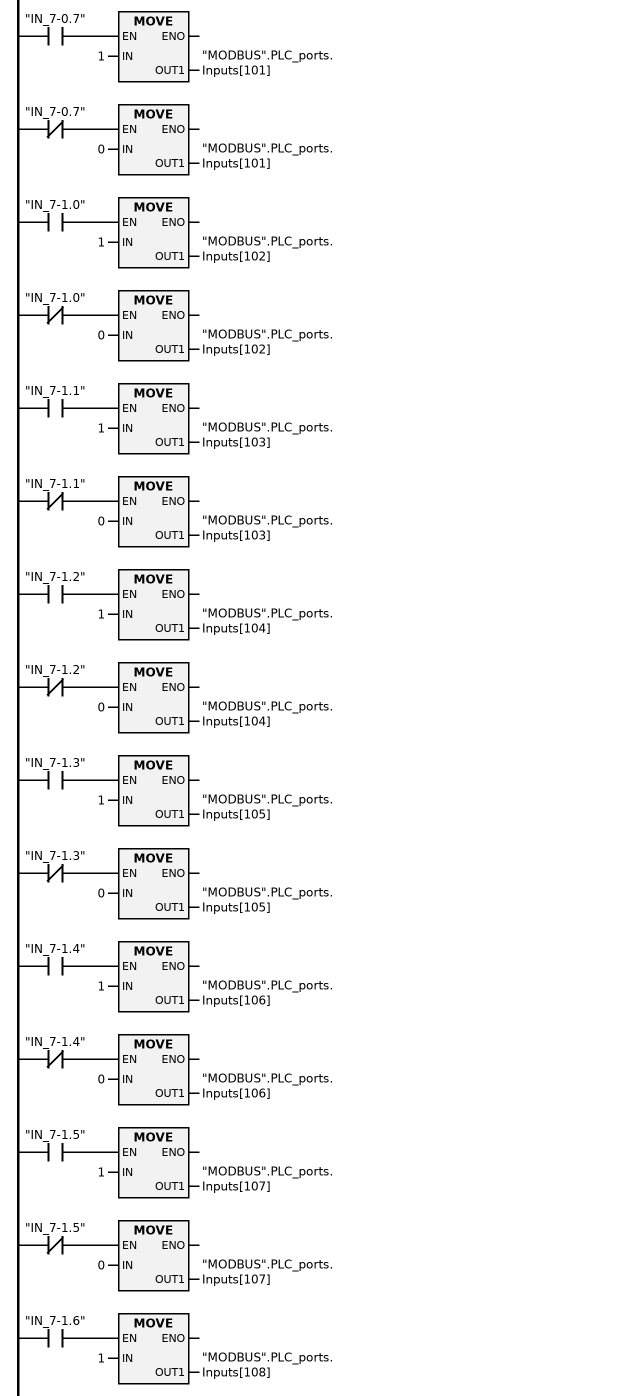
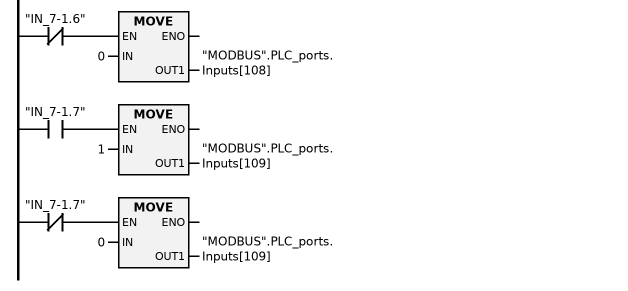
   RUNG wire#powerrail
      Contact( "IN_7-0.0" )
      Move(in := 1, out1 => "MODBUS".PLC_ports.Inputs[94])
   END_RUNG
   RUNG wire#powerrail
      I_Contact( "IN_7-0.0" )
      Move(in := 0, out1 => "MODBUS".PLC_ports.Inputs[94])
   END_RUNG
   RUNG wire#powerrail
      Contact( "IN_7-0.1" )
      Move(in := 1, out1 => "MODBUS".PLC_ports.Inputs[95])
   END_RUNG
   RUNG wire#powerrail
      I_Contact( "IN_7-0.1" )
      Move(in := 0, out1 => "MODBUS".PLC_ports.Inputs[95])
   END_RUNG
   RUNG wire#powerrail
      Contact( "IN_7-0.2" )
      Move(in := 1, out1 => "MODBUS".PLC_ports.Inputs[96])
   END_RUNG
   RUNG wire#powerrail
      I_Contact( "IN_7-0.2" )
      Move(in := 0, out1 => "MODBUS".PLC_ports.Inputs[96])
   END_RUNG
   RUNG wire#powerrail
      Contact( "IN_7-0.3" )
      Move(in := 1, out1 => "MODBUS".PLC_ports.Inputs[97])
   END_RUNG
   RUNG wire#powerrail
      I_Contact( "IN_7-0.3" )
      Move(in := 0, out1 => "MODBUS".PLC_ports.Inputs[97])
   END_RUNG
   RUNG wire#powerrail
      Contact( "IN_7-0.4" )
      Move(in := 1, out1 => "MODBUS".PLC_ports.Inputs[98])
   END_RUNG
   RUNG wire#powerrail
      I_Contact( "IN_7-0.4" )
      Move(in := 0, out1 => "MODBUS".PLC_ports.Inputs[98])
   END_RUNG
   RUNG wire#powerrail
      Contact( "IN_7-0.5" )
      Move(in := 1, out1 => "MODBUS".PLC_ports.Inputs[99])
   END_RUNG
   RUNG wire#powerrail
      I_Contact( "IN_7-0.5" )
      Move(in := 0, out1 => "MODBUS".PLC_ports.Inputs[99])
   END_RUNG
   RUNG wire#powerrail
      Contact( "IN_7-0.6" )
      Move(in := 1, out1 => "MODBUS".PLC_ports.Inputs[100])
   END_RUNG
   RUNG wire#powerrail
      I_Contact( "IN_7-0.6" )
      Move(in := 0, out1 => "MODBUS".PLC_ports.Inputs[100])
   END_RUNG
   RUNG wire#powerrail
      Contact( "IN_7-0.7" )
      Move(in := 1, out1 => "MODBUS".PLC_ports.Inputs[101])
   END_RUNG
   RUNG wire#powerrail
      I_Contact( "IN_7-0.7" )
      Move(in := 0, out1 => "MODBUS".PLC_ports.Inputs[101])
   END_RUNG
   RUNG wire#powerrail
      Contact( "IN_7-1.0" )
      Move(in := 1, out1 => "MODBUS".PLC_ports.Inputs[102])
   END_RUNG
   RUNG wire#powerrail
      I_Contact( "IN_7-1.0" )
      Move(in := 0, out1 => "MODBUS".PLC_ports.Inputs[102])
   END_RUNG
   RUNG wire#powerrail
      Contact( "IN_7-1.1" )
      Move(in := 1, out1 => "MODBUS".PLC_ports.Inputs[103])
   END_RUNG
   RUNG wire#powerrail
      I_Contact( "IN_7-1.1" )
      Move(in := 0, out1 => "MODBUS".PLC_ports.Inputs[103])
   END_RUNG
   RUNG wire#powerrail
      Contact( "IN_7-1.2" )
      Move(in := 1, out1 => "MODBUS".PLC_ports.Inputs[104])
   END_RUNG
   RUNG wire#powerrail
      I_Contact( "IN_7-1.2" )
      Move(in := 0, out1 => "MODBUS".PLC_ports.Inputs[104])
   END_RUNG
   RUNG wire#powerrail
      Contact( "IN_7-1.3" )
      Move(in := 1, out1 => "MODBUS".PLC_ports.Inputs[105])
   END_RUNG
   RUNG wire#powerrail
      I_Contact( "IN_7-1.3" )
      Move(in := 0, out1 => "MODBUS".PLC_ports.Inputs[105])
   END_RUNG
   RUNG wire#powerrail
      Contact( "IN_7-1.4" )
      Move(in := 1, out1 => "MODBUS".PLC_ports.Inputs[106])
   END_RUNG
   RUNG wire#powerrail
      I_Contact( "IN_7-1.4" )
      Move(in := 0, out1 => "MODBUS".PLC_ports.Inputs[106])
   END_RUNG
   RUNG wire#powerrail
      Contact( "IN_7-1.5" )
      Move(in := 1, out1 => "MODBUS".PLC_ports.Inputs[107])
   END_RUNG
   RUNG wire#powerrail
      I_Contact( "IN_7-1.5" )
      Move(in := 0, out1 => "MODBUS".PLC_ports.Inputs[107])
   END_RUNG
   RUNG wire#powerrail
      Contact( "IN_7-1.6" )
      Move(in := 1, out1 => "MODBUS".PLC_ports.Inputs[108])
   END_RUNG
   RUNG wire#powerrail
      I_Contact( "IN_7-1.6" )
      Move(in := 0, out1 => "MODBUS".PLC_ports.Inputs[108])
   END_RUNG
   RUNG wire#powerrail
      Contact( "IN_7-1.7" )
      Move(in := 1, out1 => "MODBUS".PLC_ports.Inputs[109])
   END_RUNG
   RUNG wire#powerrail
      I_Contact( "IN_7-1.7" )
      Move(in := 0, out1 => "MODBUS".PLC_ports.Inputs[109])
   END_RUNG
   // the same network as SCL:
   IF "IN_7-0.0" THEN "MODBUS".PLC_ports.Inputs[94] := 1; END_IF;
   IF NOT "IN_7-0.0" THEN "MODBUS".PLC_ports.Inputs[94] := 0; END_IF;
   IF "IN_7-0.1" THEN "MODBUS".PLC_ports.Inputs[95] := 1; END_IF;
   IF NOT "IN_7-0.1" THEN "MODBUS".PLC_ports.Inputs[95] := 0; END_IF;
   IF "IN_7-0.2" THEN "MODBUS".PLC_ports.Inputs[96] := 1; END_IF;
   IF NOT "IN_7-0.2" THEN "MODBUS".PLC_ports.Inputs[96] := 0; END_IF;
   IF "IN_7-0.3" THEN "MODBUS".PLC_ports.Inputs[97] := 1; END_IF;
   IF NOT "IN_7-0.3" THEN "MODBUS".PLC_ports.Inputs[97] := 0; END_IF;
   IF "IN_7-0.4" THEN "MODBUS".PLC_ports.Inputs[98] := 1; END_IF;
   IF NOT "IN_7-0.4" THEN "MODBUS".PLC_ports.Inputs[98] := 0; END_IF;
   IF "IN_7-0.5" THEN "MODBUS".PLC_ports.Inputs[99] := 1; END_IF;
   IF NOT "IN_7-0.5" THEN "MODBUS".PLC_ports.Inputs[99] := 0; END_IF;
   IF "IN_7-0.6" THEN "MODBUS".PLC_ports.Inputs[100] := 1; END_IF;
   IF NOT "IN_7-0.6" THEN "MODBUS".PLC_ports.Inputs[100] := 0; END_IF;
   IF "IN_7-0.7" THEN "MODBUS".PLC_ports.Inputs[101] := 1; END_IF;
   IF NOT "IN_7-0.7" THEN "MODBUS".PLC_ports.Inputs[101] := 0; END_IF;
   IF "IN_7-1.0" THEN "MODBUS".PLC_ports.Inputs[102] := 1; END_IF;
   IF NOT "IN_7-1.0" THEN "MODBUS".PLC_ports.Inputs[102] := 0; END_IF;
   IF "IN_7-1.1" THEN "MODBUS".PLC_ports.Inputs[103] := 1; END_IF;
   IF NOT "IN_7-1.1" THEN "MODBUS".PLC_ports.Inputs[103] := 0; END_IF;
   IF "IN_7-1.2" THEN "MODBUS".PLC_ports.Inputs[104] := 1; END_IF;
   IF NOT "IN_7-1.2" THEN "MODBUS".PLC_ports.Inputs[104] := 0; END_IF;
   IF "IN_7-1.3" THEN "MODBUS".PLC_ports.Inputs[105] := 1; END_IF;
   IF NOT "IN_7-1.3" THEN "MODBUS".PLC_ports.Inputs[105] := 0; END_IF;
   IF "IN_7-1.4" THEN "MODBUS".PLC_ports.Inputs[106] := 1; END_IF;
   IF NOT "IN_7-1.4" THEN "MODBUS".PLC_ports.Inputs[106] := 0; END_IF;
   IF "IN_7-1.5" THEN "MODBUS".PLC_ports.Inputs[107] := 1; END_IF;
   IF NOT "IN_7-1.5" THEN "MODBUS".PLC_ports.Inputs[107] := 0; END_IF;
   IF "IN_7-1.6" THEN "MODBUS".PLC_ports.Inputs[108] := 1; END_IF;
   IF NOT "IN_7-1.6" THEN "MODBUS".PLC_ports.Inputs[108] := 0; END_IF;
   IF "IN_7-1.7" THEN "MODBUS".PLC_ports.Inputs[109] := 1; END_IF;
   IF NOT "IN_7-1.7" THEN "MODBUS".PLC_ports.Inputs[109] := 0; END_IF;
END_REGION
END_FUNCTION_BLOCK

FUNCTION_BLOCK "Output signals"   // FB3, LAD
{ S7_Optimized_Access := 'TRUE' }
VERSION : 0.1
BEGIN

REGION Network 1
   // Выходы 1 блока, Siemens S7-1200
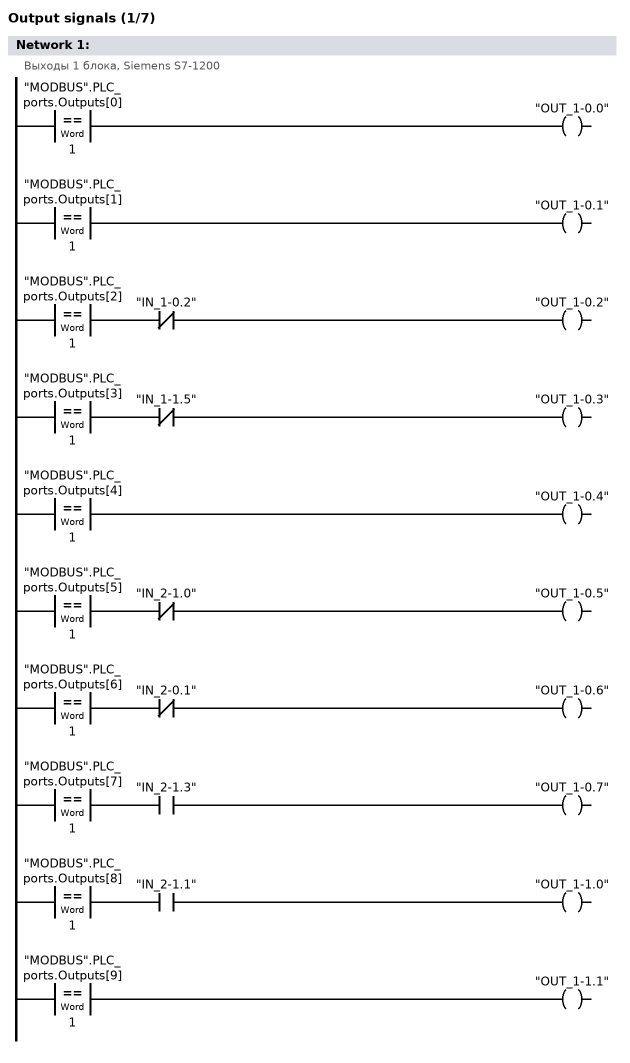
   RUNG wire#powerrail
      { S7_Templates := "SrcType := Word" } EQ_Contact(in1 := "MODBUS".PLC_ports.Outputs[0], in2 := 1)
      Coil( "OUT_1-0.0" )
   END_RUNG
   RUNG wire#powerrail
      { S7_Templates := "SrcType := Word" } EQ_Contact(in1 := "MODBUS".PLC_ports.Outputs[1], in2 := 1)
      Coil( "OUT_1-0.1" )
   END_RUNG
   RUNG wire#powerrail
      { S7_Templates := "SrcType := Word" } EQ_Contact(in1 := "MODBUS".PLC_ports.Outputs[2], in2 := 1)
      I_Contact( "IN_1-0.2" )
      Coil( "OUT_1-0.2" )
   END_RUNG
   RUNG wire#powerrail
      { S7_Templates := "SrcType := Word" } EQ_Contact(in1 := "MODBUS".PLC_ports.Outputs[3], in2 := 1)
      I_Contact( "IN_1-1.5" )
      Coil( "OUT_1-0.3" )
   END_RUNG
   RUNG wire#powerrail
      { S7_Templates := "SrcType := Word" } EQ_Contact(in1 := "MODBUS".PLC_ports.Outputs[4], in2 := 1)
      Coil( "OUT_1-0.4" )
   END_RUNG
   RUNG wire#powerrail
      { S7_Templates := "SrcType := Word" } EQ_Contact(in1 := "MODBUS".PLC_ports.Outputs[5], in2 := 1)
      I_Contact( "IN_2-1.0" )
      Coil( "OUT_1-0.5" )
   END_RUNG
   RUNG wire#powerrail
      { S7_Templates := "SrcType := Word" } EQ_Contact(in1 := "MODBUS".PLC_ports.Outputs[6], in2 := 1)
      I_Contact( "IN_2-0.1" )
      Coil( "OUT_1-0.6" )
   END_RUNG
   RUNG wire#powerrail
      { S7_Templates := "SrcType := Word" } EQ_Contact(in1 := "MODBUS".PLC_ports.Outputs[7], in2 := 1)
      Contact( "IN_2-1.3" )
      Coil( "OUT_1-0.7" )
   END_RUNG
   RUNG wire#powerrail
      { S7_Templates := "SrcType := Word" } EQ_Contact(in1 := "MODBUS".PLC_ports.Outputs[8], in2 := 1)
      Contact( "IN_2-1.1" )
      Coil( "OUT_1-1.0" )
   END_RUNG
   RUNG wire#powerrail
      { S7_Templates := "SrcType := Word" } EQ_Contact(in1 := "MODBUS".PLC_ports.Outputs[9], in2 := 1)
      Coil( "OUT_1-1.1" )
   END_RUNG
   // the same network as SCL:
   "OUT_1-0.0" := "MODBUS".PLC_ports.Outputs[0] = 1;
   "OUT_1-0.1" := "MODBUS".PLC_ports.Outputs[1] = 1;
   "OUT_1-0.2" := ("MODBUS".PLC_ports.Outputs[2] = 1) AND NOT "IN_1-0.2";
   "OUT_1-0.3" := ("MODBUS".PLC_ports.Outputs[3] = 1) AND NOT "IN_1-1.5";
   "OUT_1-0.4" := "MODBUS".PLC_ports.Outputs[4] = 1;
   "OUT_1-0.5" := ("MODBUS".PLC_ports.Outputs[5] = 1) AND NOT "IN_2-1.0";
   "OUT_1-0.6" := ("MODBUS".PLC_ports.Outputs[6] = 1) AND NOT "IN_2-0.1";
   "OUT_1-0.7" := ("MODBUS".PLC_ports.Outputs[7] = 1) AND "IN_2-1.3";
   "OUT_1-1.0" := ("MODBUS".PLC_ports.Outputs[8] = 1) AND "IN_2-1.1";
   "OUT_1-1.1" := "MODBUS".PLC_ports.Outputs[9] = 1;
END_REGION

REGION Network 2
   // Выходы 2 блока, Siemens SM-1223
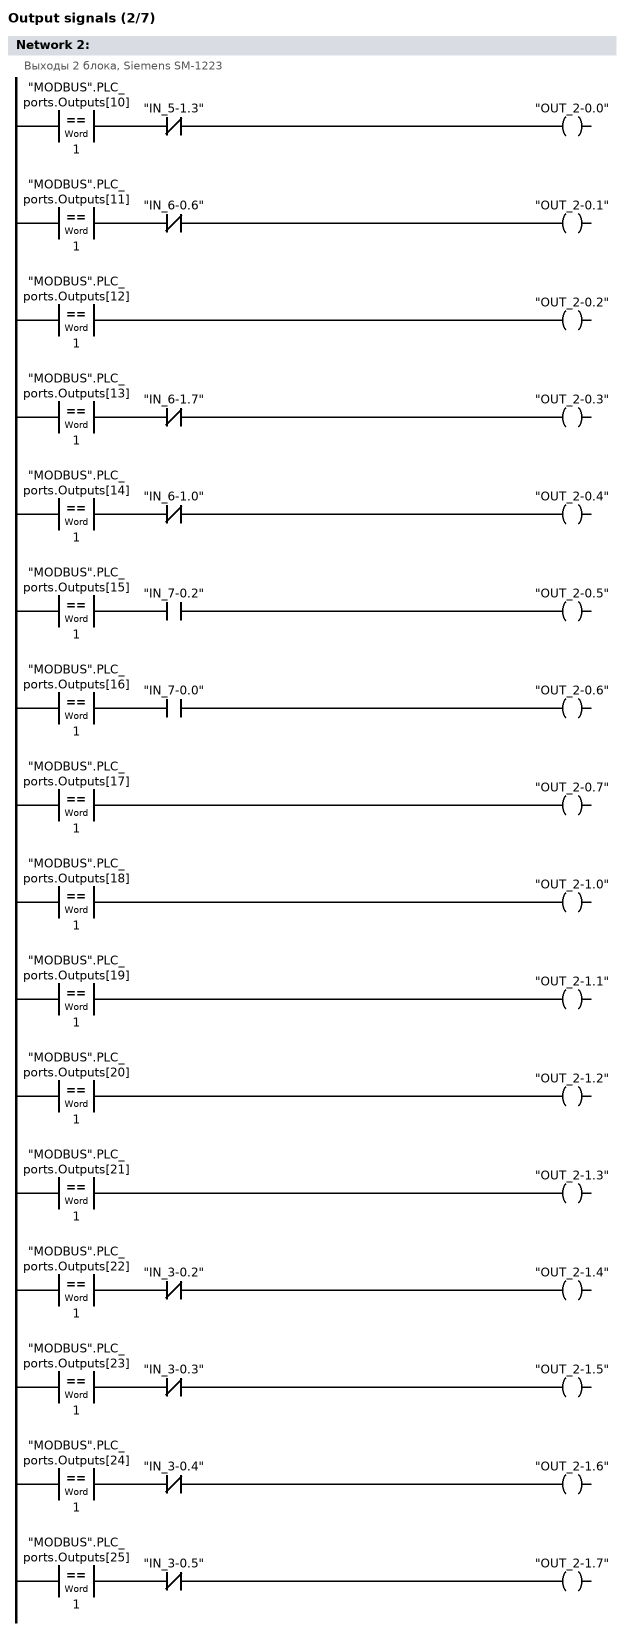
   RUNG wire#powerrail
      { S7_Templates := "SrcType := Word" } EQ_Contact(in1 := "MODBUS".PLC_ports.Outputs[10], in2 := 1)
      I_Contact( "IN_5-1.3" )
      Coil( "OUT_2-0.0" )
   END_RUNG
   RUNG wire#powerrail
      { S7_Templates := "SrcType := Word" } EQ_Contact(in1 := "MODBUS".PLC_ports.Outputs[11], in2 := 1)
      I_Contact( "IN_6-0.6" )
      Coil( "OUT_2-0.1" )
   END_RUNG
   RUNG wire#powerrail
      { S7_Templates := "SrcType := Word" } EQ_Contact(in1 := "MODBUS".PLC_ports.Outputs[12], in2 := 1)
      Coil( "OUT_2-0.2" )
   END_RUNG
   RUNG wire#powerrail
      { S7_Templates := "SrcType := Word" } EQ_Contact(in1 := "MODBUS".PLC_ports.Outputs[13], in2 := 1)
      I_Contact( "IN_6-1.7" )
      Coil( "OUT_2-0.3" )
   END_RUNG
   RUNG wire#powerrail
      { S7_Templates := "SrcType := Word" } EQ_Contact(in1 := "MODBUS".PLC_ports.Outputs[14], in2 := 1)
      I_Contact( "IN_6-1.0" )
      Coil( "OUT_2-0.4" )
   END_RUNG
   RUNG wire#powerrail
      { S7_Templates := "SrcType := Word" } EQ_Contact(in1 := "MODBUS".PLC_ports.Outputs[15], in2 := 1)
      Contact( "IN_7-0.2" )
      Coil( "OUT_2-0.5" )
   END_RUNG
   RUNG wire#powerrail
      { S7_Templates := "SrcType := Word" } EQ_Contact(in1 := "MODBUS".PLC_ports.Outputs[16], in2 := 1)
      Contact( "IN_7-0.0" )
      Coil( "OUT_2-0.6" )
   END_RUNG
   RUNG wire#powerrail
      { S7_Templates := "SrcType := Word" } EQ_Contact(in1 := "MODBUS".PLC_ports.Outputs[17], in2 := 1)
      Coil( "OUT_2-0.7" )
   END_RUNG
   RUNG wire#powerrail
      { S7_Templates := "SrcType := Word" } EQ_Contact(in1 := "MODBUS".PLC_ports.Outputs[18], in2 := 1)
      Coil( "OUT_2-1.0" )
   END_RUNG
   RUNG wire#powerrail
      { S7_Templates := "SrcType := Word" } EQ_Contact(in1 := "MODBUS".PLC_ports.Outputs[19], in2 := 1)
      Coil( "OUT_2-1.1" )
   END_RUNG
   RUNG wire#powerrail
      { S7_Templates := "SrcType := Word" } EQ_Contact(in1 := "MODBUS".PLC_ports.Outputs[20], in2 := 1)
      Coil( "OUT_2-1.2" )
   END_RUNG
   RUNG wire#powerrail
      { S7_Templates := "SrcType := Word" } EQ_Contact(in1 := "MODBUS".PLC_ports.Outputs[21], in2 := 1)
      Coil( "OUT_2-1.3" )
   END_RUNG
   RUNG wire#powerrail
      { S7_Templates := "SrcType := Word" } EQ_Contact(in1 := "MODBUS".PLC_ports.Outputs[22], in2 := 1)
      I_Contact( "IN_3-0.2" )
      Coil( "OUT_2-1.4" )
   END_RUNG
   RUNG wire#powerrail
      { S7_Templates := "SrcType := Word" } EQ_Contact(in1 := "MODBUS".PLC_ports.Outputs[23], in2 := 1)
      I_Contact( "IN_3-0.3" )
      Coil( "OUT_2-1.5" )
   END_RUNG
   RUNG wire#powerrail
      { S7_Templates := "SrcType := Word" } EQ_Contact(in1 := "MODBUS".PLC_ports.Outputs[24], in2 := 1)
      I_Contact( "IN_3-0.4" )
      Coil( "OUT_2-1.6" )
   END_RUNG
   RUNG wire#powerrail
      { S7_Templates := "SrcType := Word" } EQ_Contact(in1 := "MODBUS".PLC_ports.Outputs[25], in2 := 1)
      I_Contact( "IN_3-0.5" )
      Coil( "OUT_2-1.7" )
   END_RUNG
   // the same network as SCL:
   "OUT_2-0.0" := ("MODBUS".PLC_ports.Outputs[10] = 1) AND NOT "IN_5-1.3";
   "OUT_2-0.1" := ("MODBUS".PLC_ports.Outputs[11] = 1) AND NOT "IN_6-0.6";
   "OUT_2-0.2" := "MODBUS".PLC_ports.Outputs[12] = 1;
   "OUT_2-0.3" := ("MODBUS".PLC_ports.Outputs[13] = 1) AND NOT "IN_6-1.7";
   "OUT_2-0.4" := ("MODBUS".PLC_ports.Outputs[14] = 1) AND NOT "IN_6-1.0";
   "OUT_2-0.5" := ("MODBUS".PLC_ports.Outputs[15] = 1) AND "IN_7-0.2";
   "OUT_2-0.6" := ("MODBUS".PLC_ports.Outputs[16] = 1) AND "IN_7-0.0";
   "OUT_2-0.7" := "MODBUS".PLC_ports.Outputs[17] = 1;
   "OUT_2-1.0" := "MODBUS".PLC_ports.Outputs[18] = 1;
   "OUT_2-1.1" := "MODBUS".PLC_ports.Outputs[19] = 1;
   "OUT_2-1.2" := "MODBUS".PLC_ports.Outputs[20] = 1;
   "OUT_2-1.3" := "MODBUS".PLC_ports.Outputs[21] = 1;
   "OUT_2-1.4" := ("MODBUS".PLC_ports.Outputs[22] = 1) AND NOT "IN_3-0.2";
   "OUT_2-1.5" := ("MODBUS".PLC_ports.Outputs[23] = 1) AND NOT "IN_3-0.3";
   "OUT_2-1.6" := ("MODBUS".PLC_ports.Outputs[24] = 1) AND NOT "IN_3-0.4";
   "OUT_2-1.7" := ("MODBUS".PLC_ports.Outputs[25] = 1) AND NOT "IN_3-0.5";
END_REGION

REGION Network 3
   // Выходы 3 блока, Siemens SM-1223
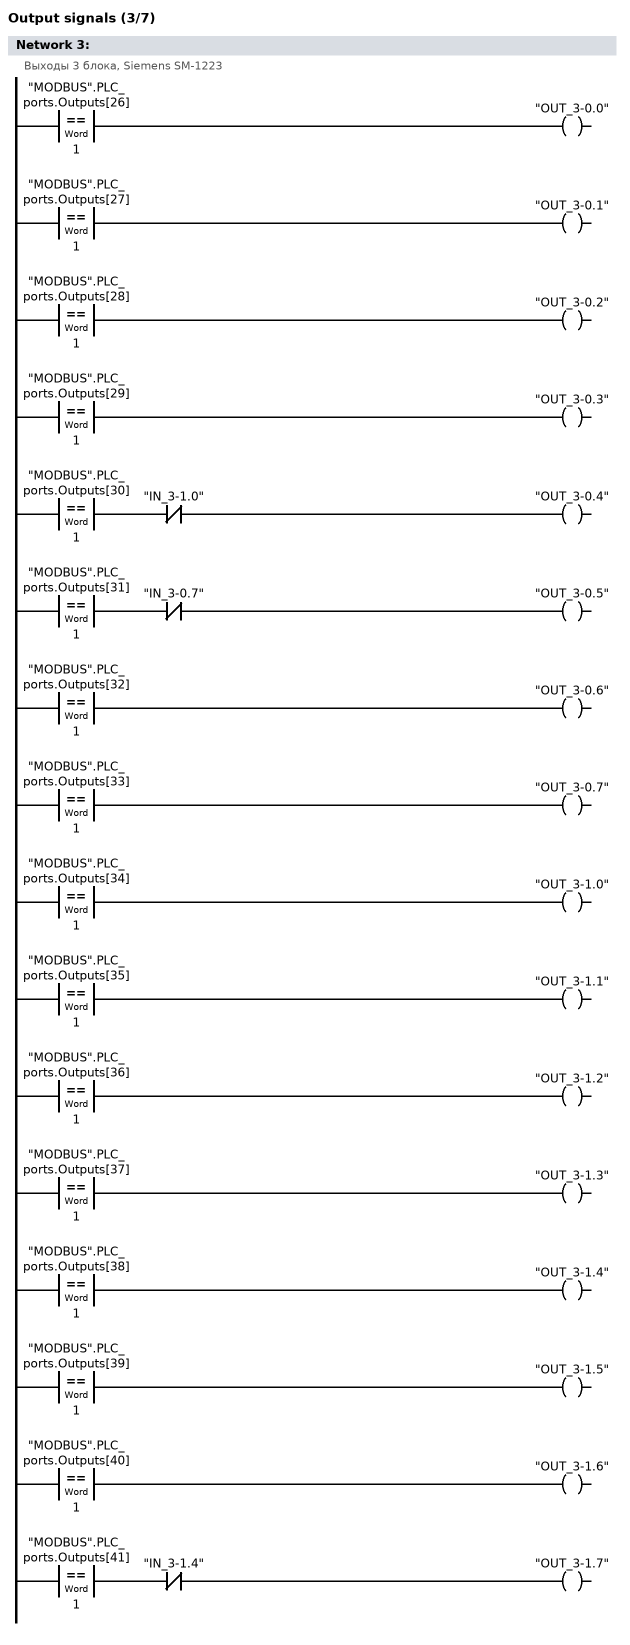
   RUNG wire#powerrail
      { S7_Templates := "SrcType := Word" } EQ_Contact(in1 := "MODBUS".PLC_ports.Outputs[26], in2 := 1)
      Coil( "OUT_3-0.0" )
   END_RUNG
   RUNG wire#powerrail
      { S7_Templates := "SrcType := Word" } EQ_Contact(in1 := "MODBUS".PLC_ports.Outputs[27], in2 := 1)
      Coil( "OUT_3-0.1" )
   END_RUNG
   RUNG wire#powerrail
      { S7_Templates := "SrcType := Word" } EQ_Contact(in1 := "MODBUS".PLC_ports.Outputs[28], in2 := 1)
      Coil( "OUT_3-0.2" )
   END_RUNG
   RUNG wire#powerrail
      { S7_Templates := "SrcType := Word" } EQ_Contact(in1 := "MODBUS".PLC_ports.Outputs[29], in2 := 1)
      Coil( "OUT_3-0.3" )
   END_RUNG
   RUNG wire#powerrail
      { S7_Templates := "SrcType := Word" } EQ_Contact(in1 := "MODBUS".PLC_ports.Outputs[30], in2 := 1)
      I_Contact( "IN_3-1.0" )
      Coil( "OUT_3-0.4" )
   END_RUNG
   RUNG wire#powerrail
      { S7_Templates := "SrcType := Word" } EQ_Contact(in1 := "MODBUS".PLC_ports.Outputs[31], in2 := 1)
      I_Contact( "IN_3-0.7" )
      Coil( "OUT_3-0.5" )
   END_RUNG
   RUNG wire#powerrail
      { S7_Templates := "SrcType := Word" } EQ_Contact(in1 := "MODBUS".PLC_ports.Outputs[32], in2 := 1)
      Coil( "OUT_3-0.6" )
   END_RUNG
   RUNG wire#powerrail
      { S7_Templates := "SrcType := Word" } EQ_Contact(in1 := "MODBUS".PLC_ports.Outputs[33], in2 := 1)
      Coil( "OUT_3-0.7" )
   END_RUNG
   RUNG wire#powerrail
      { S7_Templates := "SrcType := Word" } EQ_Contact(in1 := "MODBUS".PLC_ports.Outputs[34], in2 := 1)
      Coil( "OUT_3-1.0" )
   END_RUNG
   RUNG wire#powerrail
      { S7_Templates := "SrcType := Word" } EQ_Contact(in1 := "MODBUS".PLC_ports.Outputs[35], in2 := 1)
      Coil( "OUT_3-1.1" )
   END_RUNG
   RUNG wire#powerrail
      { S7_Templates := "SrcType := Word" } EQ_Contact(in1 := "MODBUS".PLC_ports.Outputs[36], in2 := 1)
      Coil( "OUT_3-1.2" )
   END_RUNG
   RUNG wire#powerrail
      { S7_Templates := "SrcType := Word" } EQ_Contact(in1 := "MODBUS".PLC_ports.Outputs[37], in2 := 1)
      Coil( "OUT_3-1.3" )
   END_RUNG
   RUNG wire#powerrail
      { S7_Templates := "SrcType := Word" } EQ_Contact(in1 := "MODBUS".PLC_ports.Outputs[38], in2 := 1)
      Coil( "OUT_3-1.4" )
   END_RUNG
   RUNG wire#powerrail
      { S7_Templates := "SrcType := Word" } EQ_Contact(in1 := "MODBUS".PLC_ports.Outputs[39], in2 := 1)
      Coil( "OUT_3-1.5" )
   END_RUNG
   RUNG wire#powerrail
      { S7_Templates := "SrcType := Word" } EQ_Contact(in1 := "MODBUS".PLC_ports.Outputs[40], in2 := 1)
      Coil( "OUT_3-1.6" )
   END_RUNG
   RUNG wire#powerrail
      { S7_Templates := "SrcType := Word" } EQ_Contact(in1 := "MODBUS".PLC_ports.Outputs[41], in2 := 1)
      I_Contact( "IN_3-1.4" )
      Coil( "OUT_3-1.7" )
   END_RUNG
   // the same network as SCL:
   "OUT_3-0.0" := "MODBUS".PLC_ports.Outputs[26] = 1;
   "OUT_3-0.1" := "MODBUS".PLC_ports.Outputs[27] = 1;
   "OUT_3-0.2" := "MODBUS".PLC_ports.Outputs[28] = 1;
   "OUT_3-0.3" := "MODBUS".PLC_ports.Outputs[29] = 1;
   "OUT_3-0.4" := ("MODBUS".PLC_ports.Outputs[30] = 1) AND NOT "IN_3-1.0";
   "OUT_3-0.5" := ("MODBUS".PLC_ports.Outputs[31] = 1) AND NOT "IN_3-0.7";
   "OUT_3-0.6" := "MODBUS".PLC_ports.Outputs[32] = 1;
   "OUT_3-0.7" := "MODBUS".PLC_ports.Outputs[33] = 1;
   "OUT_3-1.0" := "MODBUS".PLC_ports.Outputs[34] = 1;
   "OUT_3-1.1" := "MODBUS".PLC_ports.Outputs[35] = 1;
   "OUT_3-1.2" := "MODBUS".PLC_ports.Outputs[36] = 1;
   "OUT_3-1.3" := "MODBUS".PLC_ports.Outputs[37] = 1;
   "OUT_3-1.4" := "MODBUS".PLC_ports.Outputs[38] = 1;
   "OUT_3-1.5" := "MODBUS".PLC_ports.Outputs[39] = 1;
   "OUT_3-1.6" := "MODBUS".PLC_ports.Outputs[40] = 1;
   "OUT_3-1.7" := ("MODBUS".PLC_ports.Outputs[41] = 1) AND NOT "IN_3-1.4";
END_REGION

REGION Network 4
   // Выходы 4 блока, Siemens SM-1223
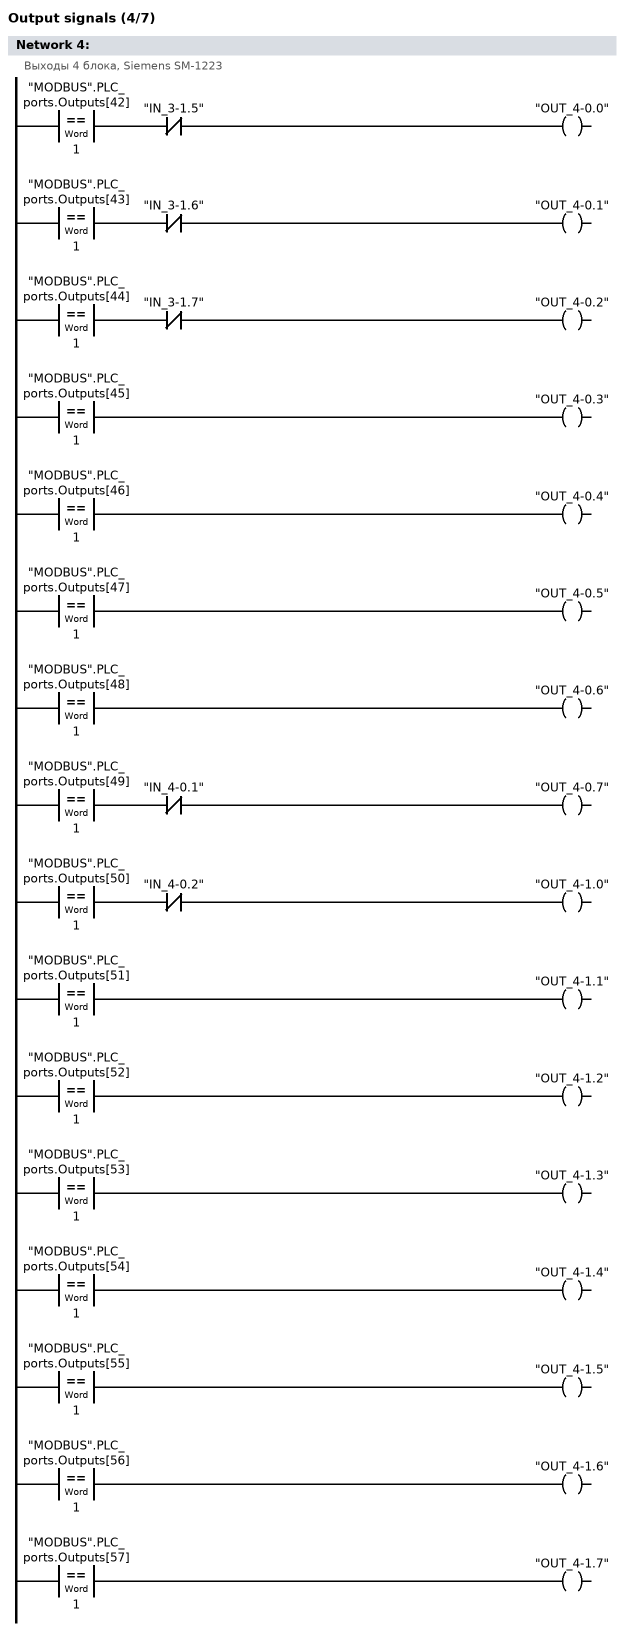
   RUNG wire#powerrail
      { S7_Templates := "SrcType := Word" } EQ_Contact(in1 := "MODBUS".PLC_ports.Outputs[42], in2 := 1)
      I_Contact( "IN_3-1.5" )
      Coil( "OUT_4-0.0" )
   END_RUNG
   RUNG wire#powerrail
      { S7_Templates := "SrcType := Word" } EQ_Contact(in1 := "MODBUS".PLC_ports.Outputs[43], in2 := 1)
      I_Contact( "IN_3-1.6" )
      Coil( "OUT_4-0.1" )
   END_RUNG
   RUNG wire#powerrail
      { S7_Templates := "SrcType := Word" } EQ_Contact(in1 := "MODBUS".PLC_ports.Outputs[44], in2 := 1)
      I_Contact( "IN_3-1.7" )
      Coil( "OUT_4-0.2" )
   END_RUNG
   RUNG wire#powerrail
      { S7_Templates := "SrcType := Word" } EQ_Contact(in1 := "MODBUS".PLC_ports.Outputs[45], in2 := 1)
      Coil( "OUT_4-0.3" )
   END_RUNG
   RUNG wire#powerrail
      { S7_Templates := "SrcType := Word" } EQ_Contact(in1 := "MODBUS".PLC_ports.Outputs[46], in2 := 1)
      Coil( "OUT_4-0.4" )
   END_RUNG
   RUNG wire#powerrail
      { S7_Templates := "SrcType := Word" } EQ_Contact(in1 := "MODBUS".PLC_ports.Outputs[47], in2 := 1)
      Coil( "OUT_4-0.5" )
   END_RUNG
   RUNG wire#powerrail
      { S7_Templates := "SrcType := Word" } EQ_Contact(in1 := "MODBUS".PLC_ports.Outputs[48], in2 := 1)
      Coil( "OUT_4-0.6" )
   END_RUNG
   RUNG wire#powerrail
      { S7_Templates := "SrcType := Word" } EQ_Contact(in1 := "MODBUS".PLC_ports.Outputs[49], in2 := 1)
      I_Contact( "IN_4-0.1" )
      Coil( "OUT_4-0.7" )
   END_RUNG
   RUNG wire#powerrail
      { S7_Templates := "SrcType := Word" } EQ_Contact(in1 := "MODBUS".PLC_ports.Outputs[50], in2 := 1)
      I_Contact( "IN_4-0.2" )
      Coil( "OUT_4-1.0" )
   END_RUNG
   RUNG wire#powerrail
      { S7_Templates := "SrcType := Word" } EQ_Contact(in1 := "MODBUS".PLC_ports.Outputs[51], in2 := 1)
      Coil( "OUT_4-1.1" )
   END_RUNG
   RUNG wire#powerrail
      { S7_Templates := "SrcType := Word" } EQ_Contact(in1 := "MODBUS".PLC_ports.Outputs[52], in2 := 1)
      Coil( "OUT_4-1.2" )
   END_RUNG
   RUNG wire#powerrail
      { S7_Templates := "SrcType := Word" } EQ_Contact(in1 := "MODBUS".PLC_ports.Outputs[53], in2 := 1)
      Coil( "OUT_4-1.3" )
   END_RUNG
   RUNG wire#powerrail
      { S7_Templates := "SrcType := Word" } EQ_Contact(in1 := "MODBUS".PLC_ports.Outputs[54], in2 := 1)
      Coil( "OUT_4-1.4" )
   END_RUNG
   RUNG wire#powerrail
      { S7_Templates := "SrcType := Word" } EQ_Contact(in1 := "MODBUS".PLC_ports.Outputs[55], in2 := 1)
      Coil( "OUT_4-1.5" )
   END_RUNG
   RUNG wire#powerrail
      { S7_Templates := "SrcType := Word" } EQ_Contact(in1 := "MODBUS".PLC_ports.Outputs[56], in2 := 1)
      Coil( "OUT_4-1.6" )
   END_RUNG
   RUNG wire#powerrail
      { S7_Templates := "SrcType := Word" } EQ_Contact(in1 := "MODBUS".PLC_ports.Outputs[57], in2 := 1)
      Coil( "OUT_4-1.7" )
   END_RUNG
   // the same network as SCL:
   "OUT_4-0.0" := ("MODBUS".PLC_ports.Outputs[42] = 1) AND NOT "IN_3-1.5";
   "OUT_4-0.1" := ("MODBUS".PLC_ports.Outputs[43] = 1) AND NOT "IN_3-1.6";
   "OUT_4-0.2" := ("MODBUS".PLC_ports.Outputs[44] = 1) AND NOT "IN_3-1.7";
   "OUT_4-0.3" := "MODBUS".PLC_ports.Outputs[45] = 1;
   "OUT_4-0.4" := "MODBUS".PLC_ports.Outputs[46] = 1;
   "OUT_4-0.5" := "MODBUS".PLC_ports.Outputs[47] = 1;
   "OUT_4-0.6" := "MODBUS".PLC_ports.Outputs[48] = 1;
   "OUT_4-0.7" := ("MODBUS".PLC_ports.Outputs[49] = 1) AND NOT "IN_4-0.1";
   "OUT_4-1.0" := ("MODBUS".PLC_ports.Outputs[50] = 1) AND NOT "IN_4-0.2";
   "OUT_4-1.1" := "MODBUS".PLC_ports.Outputs[51] = 1;
   "OUT_4-1.2" := "MODBUS".PLC_ports.Outputs[52] = 1;
   "OUT_4-1.3" := "MODBUS".PLC_ports.Outputs[53] = 1;
   "OUT_4-1.4" := "MODBUS".PLC_ports.Outputs[54] = 1;
   "OUT_4-1.5" := "MODBUS".PLC_ports.Outputs[55] = 1;
   "OUT_4-1.6" := "MODBUS".PLC_ports.Outputs[56] = 1;
   "OUT_4-1.7" := "MODBUS".PLC_ports.Outputs[57] = 1;
END_REGION

REGION Network 5
   // Выходы 5 блока, Siemens SM-1223
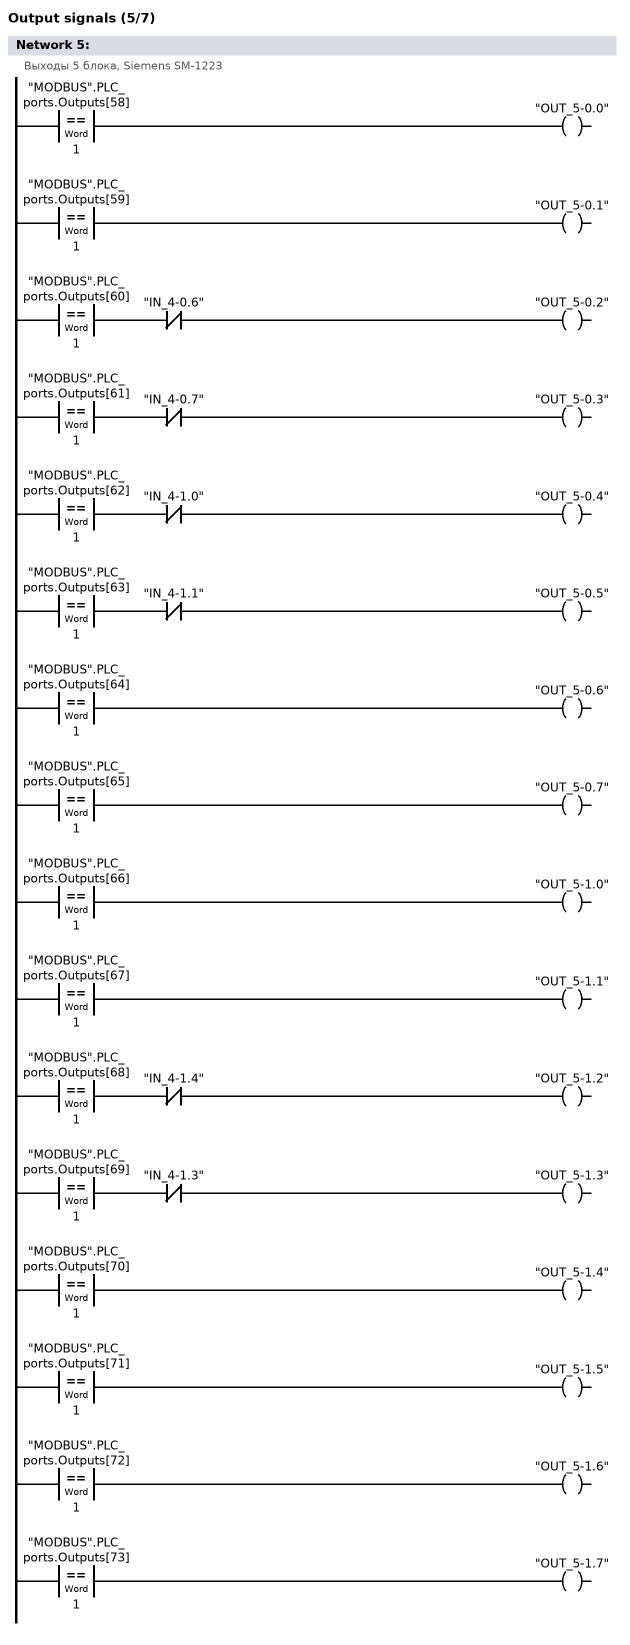
   RUNG wire#powerrail
      { S7_Templates := "SrcType := Word" } EQ_Contact(in1 := "MODBUS".PLC_ports.Outputs[58], in2 := 1)
      Coil( "OUT_5-0.0" )
   END_RUNG
   RUNG wire#powerrail
      { S7_Templates := "SrcType := Word" } EQ_Contact(in1 := "MODBUS".PLC_ports.Outputs[59], in2 := 1)
      Coil( "OUT_5-0.1" )
   END_RUNG
   RUNG wire#powerrail
      { S7_Templates := "SrcType := Word" } EQ_Contact(in1 := "MODBUS".PLC_ports.Outputs[60], in2 := 1)
      I_Contact( "IN_4-0.6" )
      Coil( "OUT_5-0.2" )
   END_RUNG
   RUNG wire#powerrail
      { S7_Templates := "SrcType := Word" } EQ_Contact(in1 := "MODBUS".PLC_ports.Outputs[61], in2 := 1)
      I_Contact( "IN_4-0.7" )
      Coil( "OUT_5-0.3" )
   END_RUNG
   RUNG wire#powerrail
      { S7_Templates := "SrcType := Word" } EQ_Contact(in1 := "MODBUS".PLC_ports.Outputs[62], in2 := 1)
      I_Contact( "IN_4-1.0" )
      Coil( "OUT_5-0.4" )
   END_RUNG
   RUNG wire#powerrail
      { S7_Templates := "SrcType := Word" } EQ_Contact(in1 := "MODBUS".PLC_ports.Outputs[63], in2 := 1)
      I_Contact( "IN_4-1.1" )
      Coil( "OUT_5-0.5" )
   END_RUNG
   RUNG wire#powerrail
      { S7_Templates := "SrcType := Word" } EQ_Contact(in1 := "MODBUS".PLC_ports.Outputs[64], in2 := 1)
      Coil( "OUT_5-0.6" )
   END_RUNG
   RUNG wire#powerrail
      { S7_Templates := "SrcType := Word" } EQ_Contact(in1 := "MODBUS".PLC_ports.Outputs[65], in2 := 1)
      Coil( "OUT_5-0.7" )
   END_RUNG
   RUNG wire#powerrail
      { S7_Templates := "SrcType := Word" } EQ_Contact(in1 := "MODBUS".PLC_ports.Outputs[66], in2 := 1)
      Coil( "OUT_5-1.0" )
   END_RUNG
   RUNG wire#powerrail
      { S7_Templates := "SrcType := Word" } EQ_Contact(in1 := "MODBUS".PLC_ports.Outputs[67], in2 := 1)
      Coil( "OUT_5-1.1" )
   END_RUNG
   RUNG wire#powerrail
      { S7_Templates := "SrcType := Word" } EQ_Contact(in1 := "MODBUS".PLC_ports.Outputs[68], in2 := 1)
      I_Contact( "IN_4-1.4" )
      Coil( "OUT_5-1.2" )
   END_RUNG
   RUNG wire#powerrail
      { S7_Templates := "SrcType := Word" } EQ_Contact(in1 := "MODBUS".PLC_ports.Outputs[69], in2 := 1)
      I_Contact( "IN_4-1.3" )
      Coil( "OUT_5-1.3" )
   END_RUNG
   RUNG wire#powerrail
      { S7_Templates := "SrcType := Word" } EQ_Contact(in1 := "MODBUS".PLC_ports.Outputs[70], in2 := 1)
      Coil( "OUT_5-1.4" )
   END_RUNG
   RUNG wire#powerrail
      { S7_Templates := "SrcType := Word" } EQ_Contact(in1 := "MODBUS".PLC_ports.Outputs[71], in2 := 1)
      Coil( "OUT_5-1.5" )
   END_RUNG
   RUNG wire#powerrail
      { S7_Templates := "SrcType := Word" } EQ_Contact(in1 := "MODBUS".PLC_ports.Outputs[72], in2 := 1)
      Coil( "OUT_5-1.6" )
   END_RUNG
   RUNG wire#powerrail
      { S7_Templates := "SrcType := Word" } EQ_Contact(in1 := "MODBUS".PLC_ports.Outputs[73], in2 := 1)
      Coil( "OUT_5-1.7" )
   END_RUNG
   // the same network as SCL:
   "OUT_5-0.0" := "MODBUS".PLC_ports.Outputs[58] = 1;
   "OUT_5-0.1" := "MODBUS".PLC_ports.Outputs[59] = 1;
   "OUT_5-0.2" := ("MODBUS".PLC_ports.Outputs[60] = 1) AND NOT "IN_4-0.6";
   "OUT_5-0.3" := ("MODBUS".PLC_ports.Outputs[61] = 1) AND NOT "IN_4-0.7";
   "OUT_5-0.4" := ("MODBUS".PLC_ports.Outputs[62] = 1) AND NOT "IN_4-1.0";
   "OUT_5-0.5" := ("MODBUS".PLC_ports.Outputs[63] = 1) AND NOT "IN_4-1.1";
   "OUT_5-0.6" := "MODBUS".PLC_ports.Outputs[64] = 1;
   "OUT_5-0.7" := "MODBUS".PLC_ports.Outputs[65] = 1;
   "OUT_5-1.0" := "MODBUS".PLC_ports.Outputs[66] = 1;
   "OUT_5-1.1" := "MODBUS".PLC_ports.Outputs[67] = 1;
   "OUT_5-1.2" := ("MODBUS".PLC_ports.Outputs[68] = 1) AND NOT "IN_4-1.4";
   "OUT_5-1.3" := ("MODBUS".PLC_ports.Outputs[69] = 1) AND NOT "IN_4-1.3";
   "OUT_5-1.4" := "MODBUS".PLC_ports.Outputs[70] = 1;
   "OUT_5-1.5" := "MODBUS".PLC_ports.Outputs[71] = 1;
   "OUT_5-1.6" := "MODBUS".PLC_ports.Outputs[72] = 1;
   "OUT_5-1.7" := "MODBUS".PLC_ports.Outputs[73] = 1;
END_REGION

REGION Network 6
   // Выходы 6 блока, Siemens SM-1223
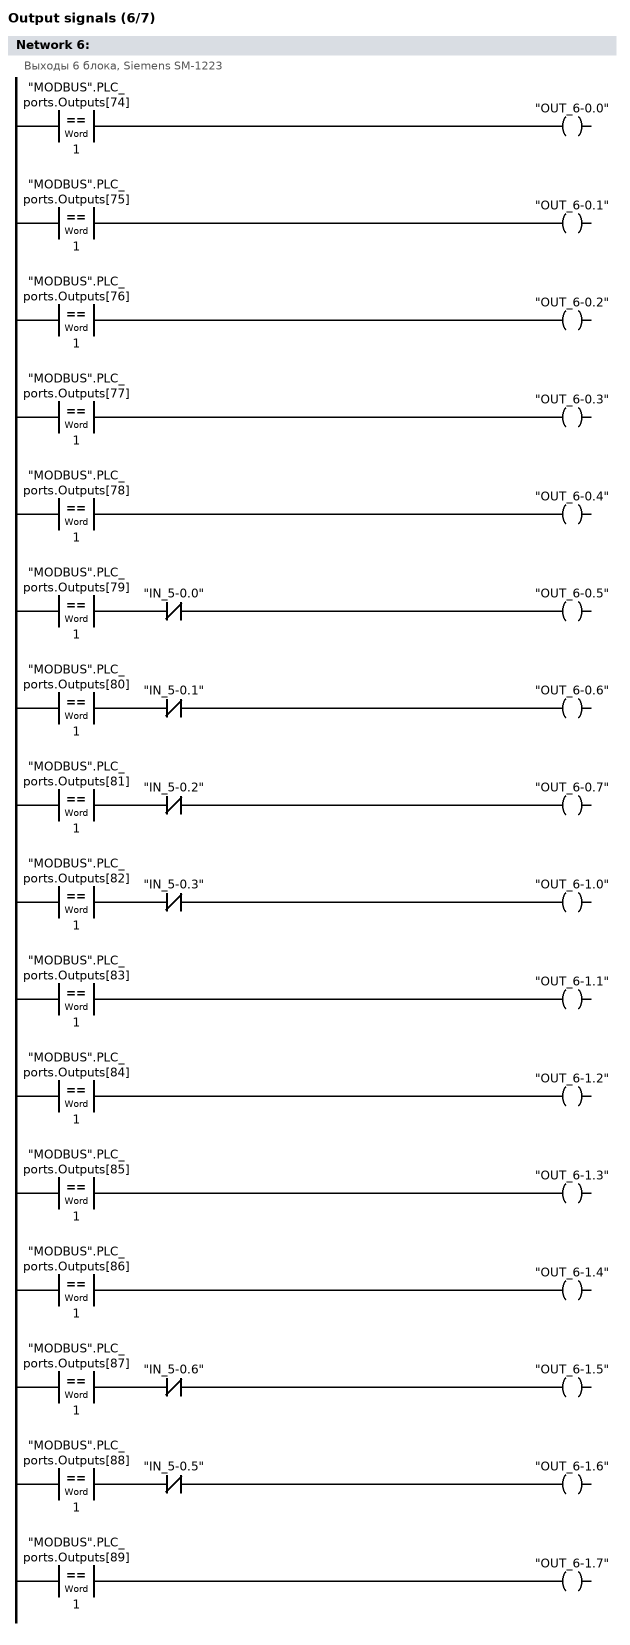
   RUNG wire#powerrail
      { S7_Templates := "SrcType := Word" } EQ_Contact(in1 := "MODBUS".PLC_ports.Outputs[74], in2 := 1)
      Coil( "OUT_6-0.0" )
   END_RUNG
   RUNG wire#powerrail
      { S7_Templates := "SrcType := Word" } EQ_Contact(in1 := "MODBUS".PLC_ports.Outputs[75], in2 := 1)
      Coil( "OUT_6-0.1" )
   END_RUNG
   RUNG wire#powerrail
      { S7_Templates := "SrcType := Word" } EQ_Contact(in1 := "MODBUS".PLC_ports.Outputs[76], in2 := 1)
      Coil( "OUT_6-0.2" )
   END_RUNG
   RUNG wire#powerrail
      { S7_Templates := "SrcType := Word" } EQ_Contact(in1 := "MODBUS".PLC_ports.Outputs[77], in2 := 1)
      Coil( "OUT_6-0.3" )
   END_RUNG
   RUNG wire#powerrail
      { S7_Templates := "SrcType := Word" } EQ_Contact(in1 := "MODBUS".PLC_ports.Outputs[78], in2 := 1)
      Coil( "OUT_6-0.4" )
   END_RUNG
   RUNG wire#powerrail
      { S7_Templates := "SrcType := Word" } EQ_Contact(in1 := "MODBUS".PLC_ports.Outputs[79], in2 := 1)
      I_Contact( "IN_5-0.0" )
      Coil( "OUT_6-0.5" )
   END_RUNG
   RUNG wire#powerrail
      { S7_Templates := "SrcType := Word" } EQ_Contact(in1 := "MODBUS".PLC_ports.Outputs[80], in2 := 1)
      I_Contact( "IN_5-0.1" )
      Coil( "OUT_6-0.6" )
   END_RUNG
   RUNG wire#powerrail
      { S7_Templates := "SrcType := Word" } EQ_Contact(in1 := "MODBUS".PLC_ports.Outputs[81], in2 := 1)
      I_Contact( "IN_5-0.2" )
      Coil( "OUT_6-0.7" )
   END_RUNG
   RUNG wire#powerrail
      { S7_Templates := "SrcType := Word" } EQ_Contact(in1 := "MODBUS".PLC_ports.Outputs[82], in2 := 1)
      I_Contact( "IN_5-0.3" )
      Coil( "OUT_6-1.0" )
   END_RUNG
   RUNG wire#powerrail
      { S7_Templates := "SrcType := Word" } EQ_Contact(in1 := "MODBUS".PLC_ports.Outputs[83], in2 := 1)
      Coil( "OUT_6-1.1" )
   END_RUNG
   RUNG wire#powerrail
      { S7_Templates := "SrcType := Word" } EQ_Contact(in1 := "MODBUS".PLC_ports.Outputs[84], in2 := 1)
      Coil( "OUT_6-1.2" )
   END_RUNG
   RUNG wire#powerrail
      { S7_Templates := "SrcType := Word" } EQ_Contact(in1 := "MODBUS".PLC_ports.Outputs[85], in2 := 1)
      Coil( "OUT_6-1.3" )
   END_RUNG
   RUNG wire#powerrail
      { S7_Templates := "SrcType := Word" } EQ_Contact(in1 := "MODBUS".PLC_ports.Outputs[86], in2 := 1)
      Coil( "OUT_6-1.4" )
   END_RUNG
   RUNG wire#powerrail
      { S7_Templates := "SrcType := Word" } EQ_Contact(in1 := "MODBUS".PLC_ports.Outputs[87], in2 := 1)
      I_Contact( "IN_5-0.6" )
      Coil( "OUT_6-1.5" )
   END_RUNG
   RUNG wire#powerrail
      { S7_Templates := "SrcType := Word" } EQ_Contact(in1 := "MODBUS".PLC_ports.Outputs[88], in2 := 1)
      I_Contact( "IN_5-0.5" )
      Coil( "OUT_6-1.6" )
   END_RUNG
   RUNG wire#powerrail
      { S7_Templates := "SrcType := Word" } EQ_Contact(in1 := "MODBUS".PLC_ports.Outputs[89], in2 := 1)
      Coil( "OUT_6-1.7" )
   END_RUNG
   // the same network as SCL:
   "OUT_6-0.0" := "MODBUS".PLC_ports.Outputs[74] = 1;
   "OUT_6-0.1" := "MODBUS".PLC_ports.Outputs[75] = 1;
   "OUT_6-0.2" := "MODBUS".PLC_ports.Outputs[76] = 1;
   "OUT_6-0.3" := "MODBUS".PLC_ports.Outputs[77] = 1;
   "OUT_6-0.4" := "MODBUS".PLC_ports.Outputs[78] = 1;
   "OUT_6-0.5" := ("MODBUS".PLC_ports.Outputs[79] = 1) AND NOT "IN_5-0.0";
   "OUT_6-0.6" := ("MODBUS".PLC_ports.Outputs[80] = 1) AND NOT "IN_5-0.1";
   "OUT_6-0.7" := ("MODBUS".PLC_ports.Outputs[81] = 1) AND NOT "IN_5-0.2";
   "OUT_6-1.0" := ("MODBUS".PLC_ports.Outputs[82] = 1) AND NOT "IN_5-0.3";
   "OUT_6-1.1" := "MODBUS".PLC_ports.Outputs[83] = 1;
   "OUT_6-1.2" := "MODBUS".PLC_ports.Outputs[84] = 1;
   "OUT_6-1.3" := "MODBUS".PLC_ports.Outputs[85] = 1;
   "OUT_6-1.4" := "MODBUS".PLC_ports.Outputs[86] = 1;
   "OUT_6-1.5" := ("MODBUS".PLC_ports.Outputs[87] = 1) AND NOT "IN_5-0.6";
   "OUT_6-1.6" := ("MODBUS".PLC_ports.Outputs[88] = 1) AND NOT "IN_5-0.5";
   "OUT_6-1.7" := "MODBUS".PLC_ports.Outputs[89] = 1;
END_REGION

REGION Network 7
   // Выходы 7 блока, Siemens SM-1223
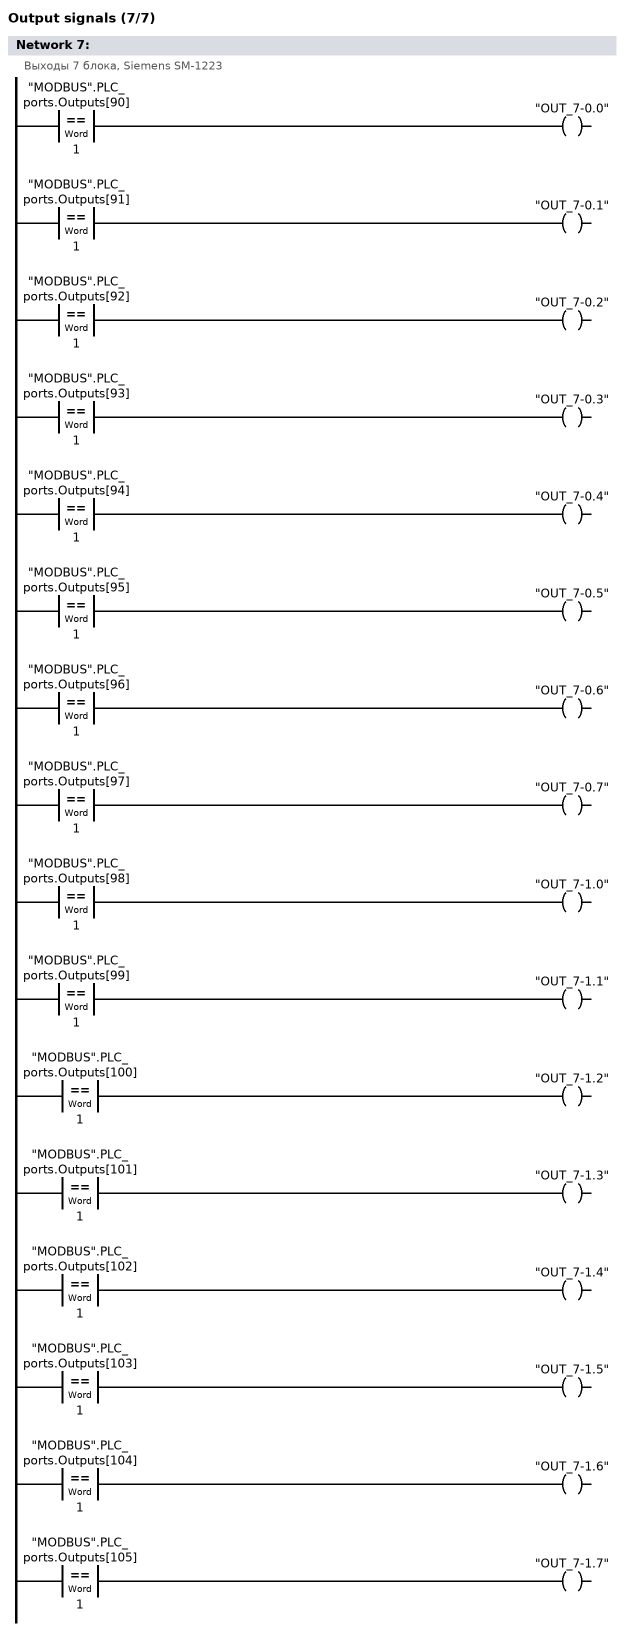
   RUNG wire#powerrail
      { S7_Templates := "SrcType := Word" } EQ_Contact(in1 := "MODBUS".PLC_ports.Outputs[90], in2 := 1)
      Coil( "OUT_7-0.0" )
   END_RUNG
   RUNG wire#powerrail
      { S7_Templates := "SrcType := Word" } EQ_Contact(in1 := "MODBUS".PLC_ports.Outputs[91], in2 := 1)
      Coil( "OUT_7-0.1" )
   END_RUNG
   RUNG wire#powerrail
      { S7_Templates := "SrcType := Word" } EQ_Contact(in1 := "MODBUS".PLC_ports.Outputs[92], in2 := 1)
      Coil( "OUT_7-0.2" )
   END_RUNG
   RUNG wire#powerrail
      { S7_Templates := "SrcType := Word" } EQ_Contact(in1 := "MODBUS".PLC_ports.Outputs[93], in2 := 1)
      Coil( "OUT_7-0.3" )
   END_RUNG
   RUNG wire#powerrail
      { S7_Templates := "SrcType := Word" } EQ_Contact(in1 := "MODBUS".PLC_ports.Outputs[94], in2 := 1)
      Coil( "OUT_7-0.4" )
   END_RUNG
   RUNG wire#powerrail
      { S7_Templates := "SrcType := Word" } EQ_Contact(in1 := "MODBUS".PLC_ports.Outputs[95], in2 := 1)
      Coil( "OUT_7-0.5" )
   END_RUNG
   RUNG wire#powerrail
      { S7_Templates := "SrcType := Word" } EQ_Contact(in1 := "MODBUS".PLC_ports.Outputs[96], in2 := 1)
      Coil( "OUT_7-0.6" )
   END_RUNG
   RUNG wire#powerrail
      { S7_Templates := "SrcType := Word" } EQ_Contact(in1 := "MODBUS".PLC_ports.Outputs[97], in2 := 1)
      Coil( "OUT_7-0.7" )
   END_RUNG
   RUNG wire#powerrail
      { S7_Templates := "SrcType := Word" } EQ_Contact(in1 := "MODBUS".PLC_ports.Outputs[98], in2 := 1)
      Coil( "OUT_7-1.0" )
   END_RUNG
   RUNG wire#powerrail
      { S7_Templates := "SrcType := Word" } EQ_Contact(in1 := "MODBUS".PLC_ports.Outputs[99], in2 := 1)
      Coil( "OUT_7-1.1" )
   END_RUNG
   RUNG wire#powerrail
      { S7_Templates := "SrcType := Word" } EQ_Contact(in1 := "MODBUS".PLC_ports.Outputs[100], in2 := 1)
      Coil( "OUT_7-1.2" )
   END_RUNG
   RUNG wire#powerrail
      { S7_Templates := "SrcType := Word" } EQ_Contact(in1 := "MODBUS".PLC_ports.Outputs[101], in2 := 1)
      Coil( "OUT_7-1.3" )
   END_RUNG
   RUNG wire#powerrail
      { S7_Templates := "SrcType := Word" } EQ_Contact(in1 := "MODBUS".PLC_ports.Outputs[102], in2 := 1)
      Coil( "OUT_7-1.4" )
   END_RUNG
   RUNG wire#powerrail
      { S7_Templates := "SrcType := Word" } EQ_Contact(in1 := "MODBUS".PLC_ports.Outputs[103], in2 := 1)
      Coil( "OUT_7-1.5" )
   END_RUNG
   RUNG wire#powerrail
      { S7_Templates := "SrcType := Word" } EQ_Contact(in1 := "MODBUS".PLC_ports.Outputs[104], in2 := 1)
      Coil( "OUT_7-1.6" )
   END_RUNG
   RUNG wire#powerrail
      { S7_Templates := "SrcType := Word" } EQ_Contact(in1 := "MODBUS".PLC_ports.Outputs[105], in2 := 1)
      Coil( "OUT_7-1.7" )
   END_RUNG
   // the same network as SCL:
   "OUT_7-0.0" := "MODBUS".PLC_ports.Outputs[90] = 1;
   "OUT_7-0.1" := "MODBUS".PLC_ports.Outputs[91] = 1;
   "OUT_7-0.2" := "MODBUS".PLC_ports.Outputs[92] = 1;
   "OUT_7-0.3" := "MODBUS".PLC_ports.Outputs[93] = 1;
   "OUT_7-0.4" := "MODBUS".PLC_ports.Outputs[94] = 1;
   "OUT_7-0.5" := "MODBUS".PLC_ports.Outputs[95] = 1;
   "OUT_7-0.6" := "MODBUS".PLC_ports.Outputs[96] = 1;
   "OUT_7-0.7" := "MODBUS".PLC_ports.Outputs[97] = 1;
   "OUT_7-1.0" := "MODBUS".PLC_ports.Outputs[98] = 1;
   "OUT_7-1.1" := "MODBUS".PLC_ports.Outputs[99] = 1;
   "OUT_7-1.2" := "MODBUS".PLC_ports.Outputs[100] = 1;
   "OUT_7-1.3" := "MODBUS".PLC_ports.Outputs[101] = 1;
   "OUT_7-1.4" := "MODBUS".PLC_ports.Outputs[102] = 1;
   "OUT_7-1.5" := "MODBUS".PLC_ports.Outputs[103] = 1;
   "OUT_7-1.6" := "MODBUS".PLC_ports.Outputs[104] = 1;
   "OUT_7-1.7" := "MODBUS".PLC_ports.Outputs[105] = 1;
END_REGION
END_FUNCTION_BLOCK